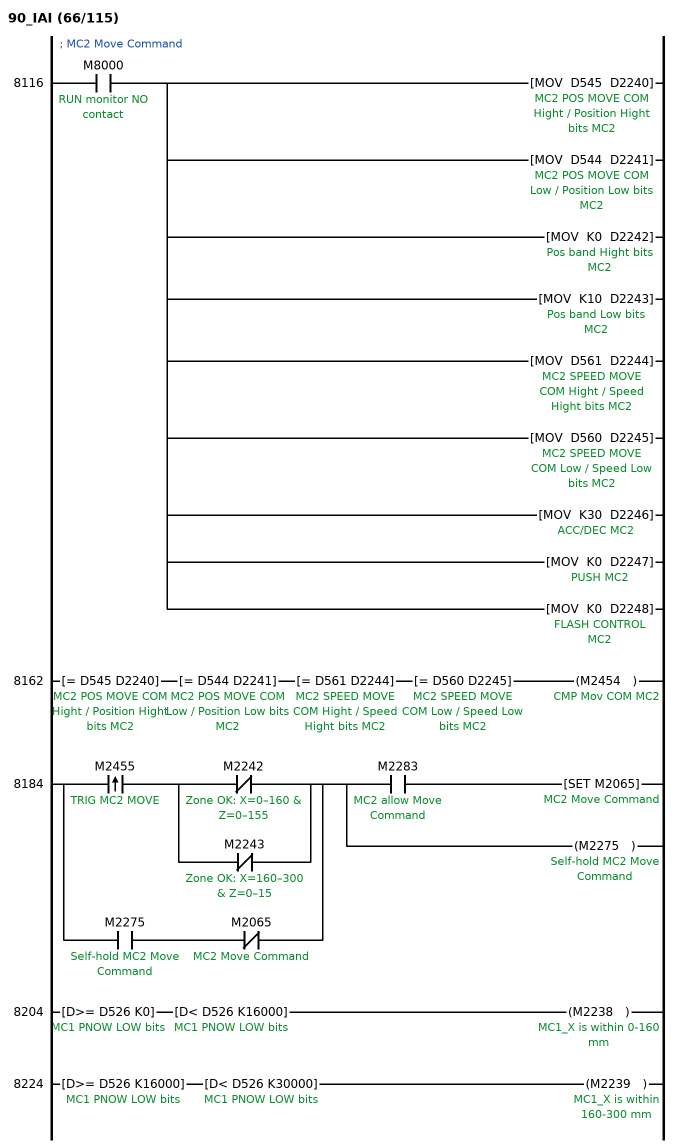
[picture p168: ladder of 90_IAI, rungs at steps 8116 to 8224]
; MC2 Move Command
8116  LD      M8000  ; RUN monitor NO contact
      MOV     D545 D2240  ; MC2 POS MOVE COM Hight / Position Hight bits MC2
      MOV     D544 D2241  ; MC2 POS MOVE COM Low / Position Low bits MC2
      MOV     K0 D2242  ; Pos band Hight bits MC2
      MOV     K10 D2243  ; Pos band Low bits MC2
      MOV     D561 D2244  ; MC2 SPEED MOVE COM Hight / Speed Hight bits MC2
      MOV     D560 D2245  ; MC2 SPEED MOVE COM Low / Speed Low bits MC2
      MOV     K30 D2246  ; ACC/DEC MC2
      MOV     K0 D2247  ; PUSH MC2
      MOV     K0 D2248  ; FLASH CONTROL MC2
8162  LD=     D545 D2240  ; MC2 POS MOVE COM Hight / Position Hight bits MC2
      AND=    D544 D2241  ; MC2 POS MOVE COM Low / Position Low bits MC2
      AND=    D561 D2244  ; MC2 SPEED MOVE COM Hight / Speed Hight bits MC2
      AND=    D560 D2245  ; MC2 SPEED MOVE COM Low / Speed Low bits MC2
      OUT     M2454  ; CMP Mov COM MC2
8184  LDP     M2455  ; TRIG MC2 MOVE
      LDI     M2242  ; Zone OK: X=0–160 & Z=0–155
      ORI     M2243  ; Zone OK: X=160–300 & Z=0–15
      ANB
      LD      M2275  ; Self-hold MC2 Move Command
      ANI     M2065  ; MC2 Move Command
      ORB
      MPS
      AND     M2283  ; MC2 allow Move Command
      SET     M2065  ; MC2 Move Command
      MPP
      OUT     M2275  ; Self-hold MC2 Move Command
8204  LDD>=   D526 K0  ; MC1 PNOW LOW bits
      ANDD<   D526 K16000  ; MC1 PNOW LOW bits
      OUT     M2238  ; MC1_X is within 0-160 mm
8224  LDD>=   D526 K16000  ; MC1 PNOW LOW bits
      ANDD<   D526 K30000  ; MC1 PNOW LOW bits
      OUT     M2239  ; MC1_X is within 160-300 mm
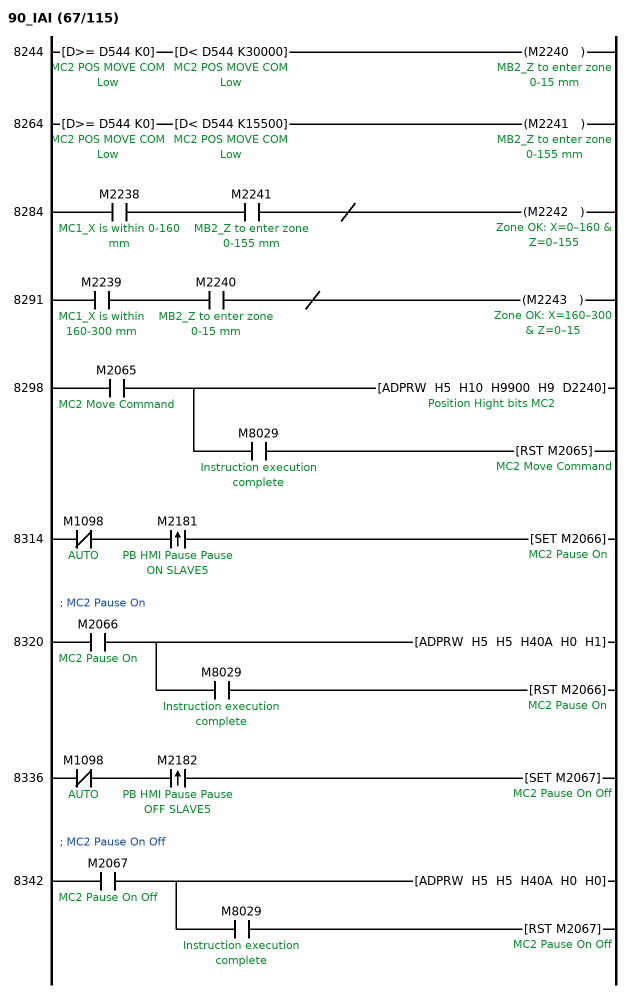
8244  LDD>=   D544 K0  ; MC2 POS MOVE COM Low
      ANDD<   D544 K30000  ; MC2 POS MOVE COM Low
      OUT     M2240  ; MB2_Z to enter zone 0-15 mm
8264  LDD>=   D544 K0  ; MC2 POS MOVE COM Low
      ANDD<   D544 K15500  ; MC2 POS MOVE COM Low
      OUT     M2241  ; MB2_Z to enter zone 0-155 mm
8284  LD      M2238  ; MC1_X is within 0-160 mm
      AND     M2241  ; MB2_Z to enter zone 0-155 mm
      INV
      OUT     M2242  ; Zone OK: X=0–160 & Z=0–155
8291  LD      M2239  ; MC1_X is within 160-300 mm
      AND     M2240  ; MB2_Z to enter zone 0-15 mm
      INV
      OUT     M2243  ; Zone OK: X=160–300 & Z=0–15
8298  LD      M2065  ; MC2 Move Command
      ADPRW   H5 H10 H9900 H9 D2240
      AND     M8029  ; Instruction execution complete
      RST     M2065  ; MC2 Move Command
8314  LDI     M1098  ; AUTO
      ANDP    M2181  ; PB HMI Pause Pause ON SLAVE5
      SET     M2066  ; MC2 Pause On
; MC2 Pause On
8320  LD      M2066  ; MC2 Pause On
      ADPRW   H5 H5 H40A H0 H1
      AND     M8029  ; Instruction execution complete
      RST     M2066  ; MC2 Pause On
8336  LDI     M1098  ; AUTO
      ANDP    M2182  ; PB HMI Pause Pause OFF SLAVE5
      SET     M2067  ; MC2 Pause On Off
; MC2 Pause On Off
8342  LD      M2067  ; MC2 Pause On Off
      ADPRW   H5 H5 H40A H0 H0
      AND     M8029  ; Instruction execution complete
      RST     M2067  ; MC2 Pause On Off
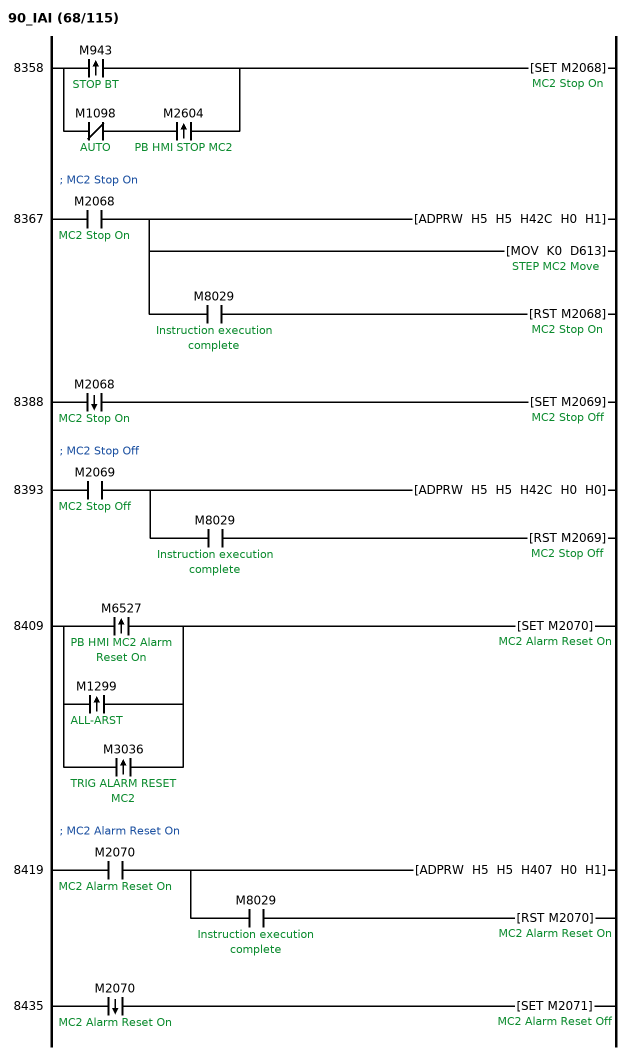
8358  LDP     M943  ; STOP BT
      LDI     M1098  ; AUTO
      ANDP    M2604  ; PB HMI STOP MC2
      ORB
      SET     M2068  ; MC2 Stop On
; MC2 Stop On
8367  LD      M2068  ; MC2 Stop On
      ADPRW   H5 H5 H42C H0 H1
      MOV     K0 D613  ; STEP MC2 Move
      AND     M8029  ; Instruction execution complete
      RST     M2068  ; MC2 Stop On
8388  LDF     M2068  ; MC2 Stop On
      SET     M2069  ; MC2 Stop Off
; MC2 Stop Off
8393  LD      M2069  ; MC2 Stop Off
      ADPRW   H5 H5 H42C H0 H0
      AND     M8029  ; Instruction execution complete
      RST     M2069  ; MC2 Stop Off
8409  LDP     M6527  ; PB HMI MC2 Alarm Reset On
      ORP     M1299  ; ALL-ARST
      ORP     M3036  ; TRIG ALARM RESET MC2
      SET     M2070  ; MC2 Alarm Reset On
; MC2 Alarm Reset On
8419  LD      M2070  ; MC2 Alarm Reset On
      ADPRW   H5 H5 H407 H0 H1
      AND     M8029  ; Instruction execution complete
      RST     M2070  ; MC2 Alarm Reset On
8435  LDF     M2070  ; MC2 Alarm Reset On
      SET     M2071  ; MC2 Alarm Reset Off
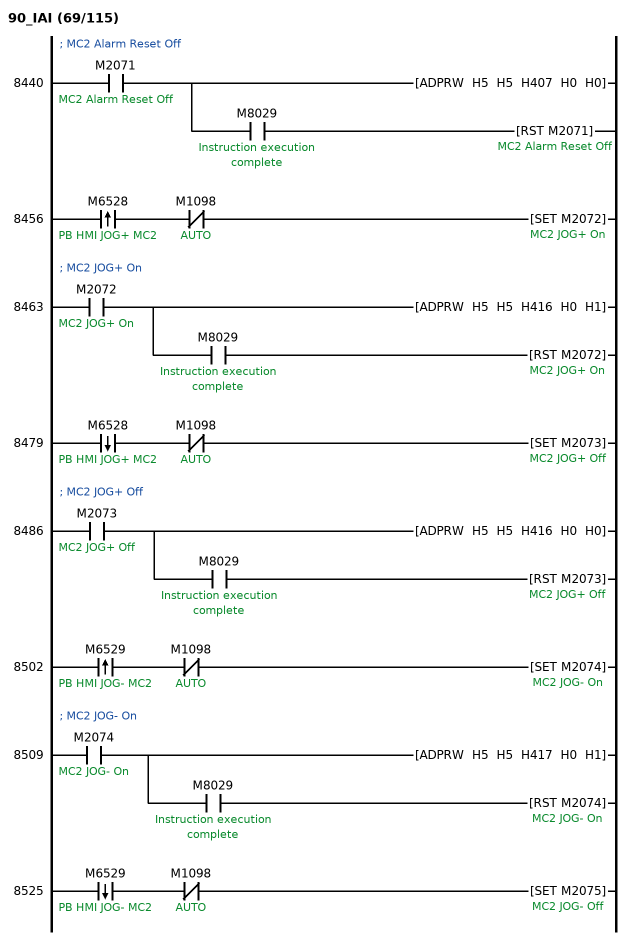
; MC2 Alarm Reset Off
8440  LD      M2071  ; MC2 Alarm Reset Off
      ADPRW   H5 H5 H407 H0 H0
      AND     M8029  ; Instruction execution complete
      RST     M2071  ; MC2 Alarm Reset Off
8456  LDP     M6528  ; PB HMI JOG+ MC2
      ANI     M1098  ; AUTO
      SET     M2072  ; MC2 JOG+ On
; MC2 JOG+ On
8463  LD      M2072  ; MC2 JOG+ On
      ADPRW   H5 H5 H416 H0 H1
      AND     M8029  ; Instruction execution complete
      RST     M2072  ; MC2 JOG+ On
8479  LDF     M6528  ; PB HMI JOG+ MC2
      ANI     M1098  ; AUTO
      SET     M2073  ; MC2 JOG+ Off
; MC2 JOG+ Off
8486  LD      M2073  ; MC2 JOG+ Off
      ADPRW   H5 H5 H416 H0 H0
      AND     M8029  ; Instruction execution complete
      RST     M2073  ; MC2 JOG+ Off
8502  LDP     M6529  ; PB HMI JOG- MC2
      ANI     M1098  ; AUTO
      SET     M2074  ; MC2 JOG- On
; MC2 JOG- On
8509  LD      M2074  ; MC2 JOG- On
      ADPRW   H5 H5 H417 H0 H1
      AND     M8029  ; Instruction execution complete
      RST     M2074  ; MC2 JOG- On
8525  LDF     M6529  ; PB HMI JOG- MC2
      ANI     M1098  ; AUTO
      SET     M2075  ; MC2 JOG- Off
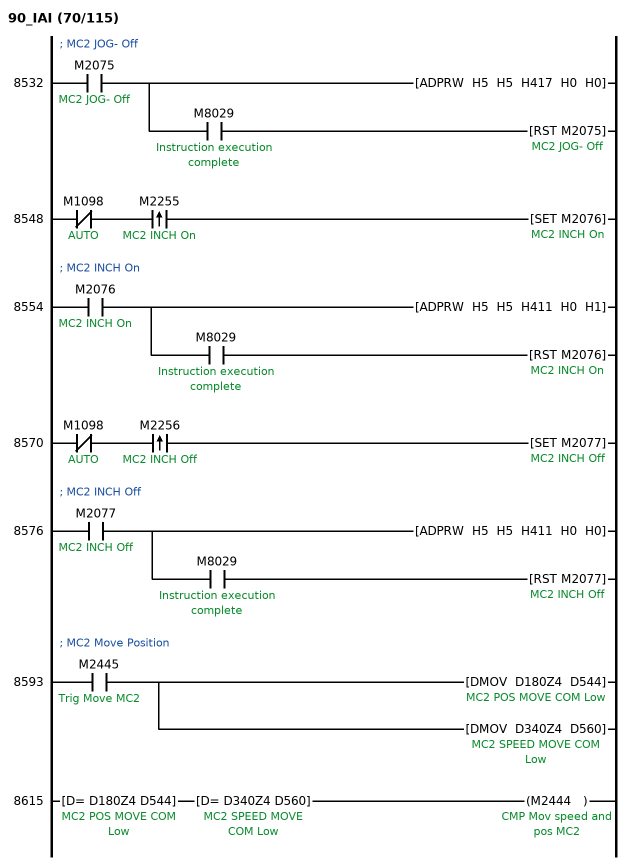
; MC2 JOG- Off
8532  LD      M2075  ; MC2 JOG- Off
      ADPRW   H5 H5 H417 H0 H0
      AND     M8029  ; Instruction execution complete
      RST     M2075  ; MC2 JOG- Off
8548  LDI     M1098  ; AUTO
      ANDP    M2255  ; MC2 INCH On
      SET     M2076  ; MC2 INCH On
; MC2 INCH On
8554  LD      M2076  ; MC2 INCH On
      ADPRW   H5 H5 H411 H0 H1
      AND     M8029  ; Instruction execution complete
      RST     M2076  ; MC2 INCH On
8570  LDI     M1098  ; AUTO
      ANDP    M2256  ; MC2 INCH Off
      SET     M2077  ; MC2 INCH Off
; MC2 INCH Off
8576  LD      M2077  ; MC2 INCH Off
      ADPRW   H5 H5 H411 H0 H0
      AND     M8029  ; Instruction execution complete
      RST     M2077  ; MC2 INCH Off
; MC2 Move Position
8593  LD      M2445  ; Trig Move MC2
      DMOV    D180Z4 D544
        [note] Position
      DMOV    D340Z4 D560
        [note] Speed
8615  LDD=    D180Z4 D544  ; MC2 POS MOVE COM Low
      ANDD=   D340Z4 D560  ; MC2 SPEED MOVE COM Low
      OUT     M2444  ; CMP Mov speed and pos MC2
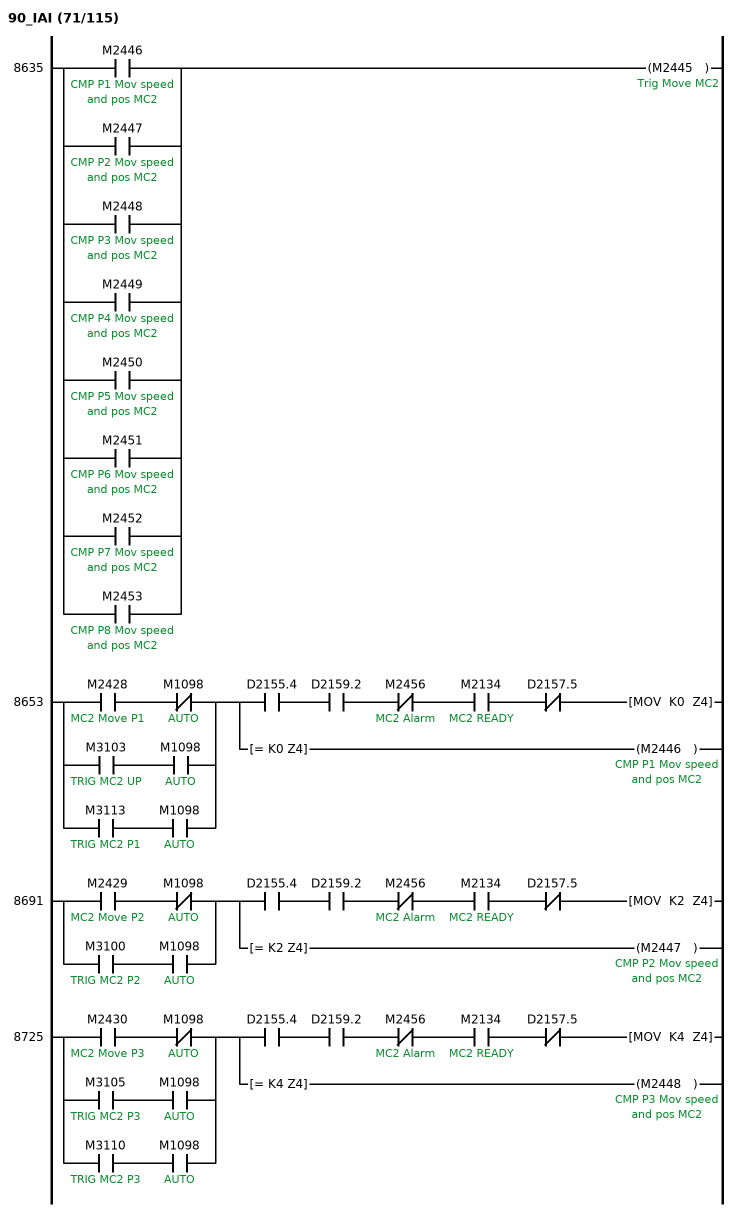
8635  LD      M2446  ; CMP P1 Mov speed and pos MC2
      OR      M2447  ; CMP P2 Mov speed and pos MC2
      OR      M2448  ; CMP P3 Mov speed and pos MC2
      OR      M2449  ; CMP P4 Mov speed and pos MC2
      OR      M2450  ; CMP P5 Mov speed and pos MC2
      OR      M2451  ; CMP P6 Mov speed and pos MC2
      OR      M2452  ; CMP P7 Mov speed and pos MC2
      OR      M2453  ; CMP P8 Mov speed and pos MC2
      OUT     M2445  ; Trig Move MC2
8653  LD      M2428  ; MC2 Move P1
      ANI     M1098  ; AUTO
      LD      M3103  ; TRIG MC2 UP
      AND     M1098  ; AUTO
      ORB
      LD      M3113  ; TRIG MC2 P1
      AND     M1098  ; AUTO
      ORB
      MPS
      AND     D2155.4
      AND     D2159.2
      ANI     M2456  ; MC2 Alarm
      AND     M2134  ; MC2 READY
      ANI     D2157.5
      MOV     K0 Z4
      MPP
      AND=    K0 Z4
      OUT     M2446  ; CMP P1 Mov speed and pos MC2
8691  LD      M2429  ; MC2 Move P2
      ANI     M1098  ; AUTO
      LD      M3100  ; TRIG MC2 P2
      AND     M1098  ; AUTO
      ORB
      MPS
      AND     D2155.4
      AND     D2159.2
      ANI     M2456  ; MC2 Alarm
      AND     M2134  ; MC2 READY
      ANI     D2157.5
      MOV     K2 Z4
      MPP
      AND=    K2 Z4
      OUT     M2447  ; CMP P2 Mov speed and pos MC2
8725  LD      M2430  ; MC2 Move P3
      ANI     M1098  ; AUTO
      LD      M3105  ; TRIG MC2 P3
      AND     M1098  ; AUTO
      ORB
      LD      M3110  ; TRIG MC2 P3
      AND     M1098  ; AUTO
      ORB
      MPS
      AND     D2155.4
      AND     D2159.2
      ANI     M2456  ; MC2 Alarm
      AND     M2134  ; MC2 READY
      ANI     D2157.5
      MOV     K4 Z4
      MPP
      AND=    K4 Z4
      OUT     M2448  ; CMP P3 Mov speed and pos MC2
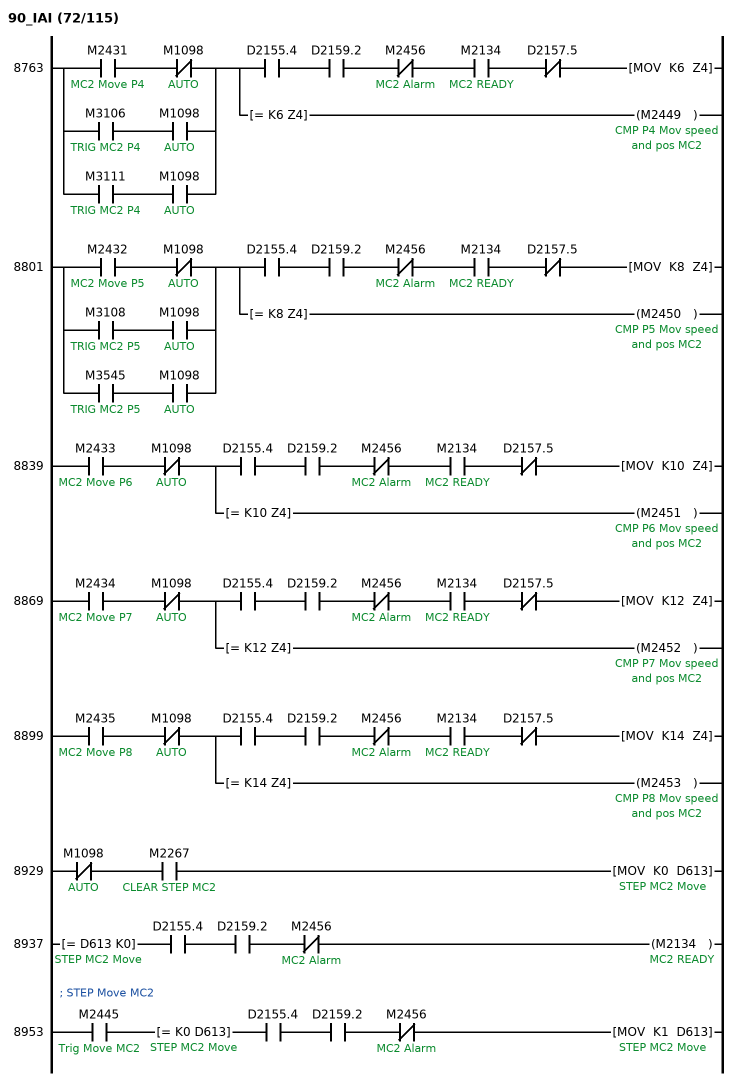
8763  LD      M2431  ; MC2 Move P4
      ANI     M1098  ; AUTO
      LD      M3106  ; TRIG MC2 P4
      AND     M1098  ; AUTO
      ORB
      LD      M3111  ; TRIG MC2 P4
      AND     M1098  ; AUTO
      ORB
      MPS
      AND     D2155.4
      AND     D2159.2
      ANI     M2456  ; MC2 Alarm
      AND     M2134  ; MC2 READY
      ANI     D2157.5
      MOV     K6 Z4
      MPP
      AND=    K6 Z4
      OUT     M2449  ; CMP P4 Mov speed and pos MC2
8801  LD      M2432  ; MC2 Move P5
      ANI     M1098  ; AUTO
      LD      M3108  ; TRIG MC2 P5
      AND     M1098  ; AUTO
      ORB
      LD      M3545  ; TRIG MC2 P5
      AND     M1098  ; AUTO
      ORB
      MPS
      AND     D2155.4
      AND     D2159.2
      ANI     M2456  ; MC2 Alarm
      AND     M2134  ; MC2 READY
      ANI     D2157.5
      MOV     K8 Z4
      MPP
      AND=    K8 Z4
      OUT     M2450  ; CMP P5 Mov speed and pos MC2
8839  LD      M2433  ; MC2 Move P6
      ANI     M1098  ; AUTO
      MPS
      AND     D2155.4
      AND     D2159.2
      ANI     M2456  ; MC2 Alarm
      AND     M2134  ; MC2 READY
      ANI     D2157.5
      MOV     K10 Z4
      MPP
      AND=    K10 Z4
      OUT     M2451  ; CMP P6 Mov speed and pos MC2
8869  LD      M2434  ; MC2 Move P7
      ANI     M1098  ; AUTO
      MPS
      AND     D2155.4
      AND     D2159.2
      ANI     M2456  ; MC2 Alarm
      AND     M2134  ; MC2 READY
      ANI     D2157.5
      MOV     K12 Z4
      MPP
      AND=    K12 Z4
      OUT     M2452  ; CMP P7 Mov speed and pos MC2
8899  LD      M2435  ; MC2 Move P8
      ANI     M1098  ; AUTO
      MPS
      AND     D2155.4
      AND     D2159.2
      ANI     M2456  ; MC2 Alarm
      AND     M2134  ; MC2 READY
      ANI     D2157.5
      MOV     K14 Z4
      MPP
      AND=    K14 Z4
      OUT     M2453  ; CMP P8 Mov speed and pos MC2
8929  LDI     M1098  ; AUTO
      AND     M2267  ; CLEAR STEP MC2
      MOV     K0 D613
8937  LD=     D613 K0  ; STEP MC2 Move
      AND     D2155.4
      AND     D2159.2
      ANI     M2456  ; MC2 Alarm
      OUT     M2134  ; MC2 READY
; STEP Move MC2
8953  LD      M2445  ; Trig Move MC2
      AND=    K0 D613  ; STEP MC2 Move
      AND     D2155.4
      AND     D2159.2
      ANI     M2456  ; MC2 Alarm
      MOV     K1 D613
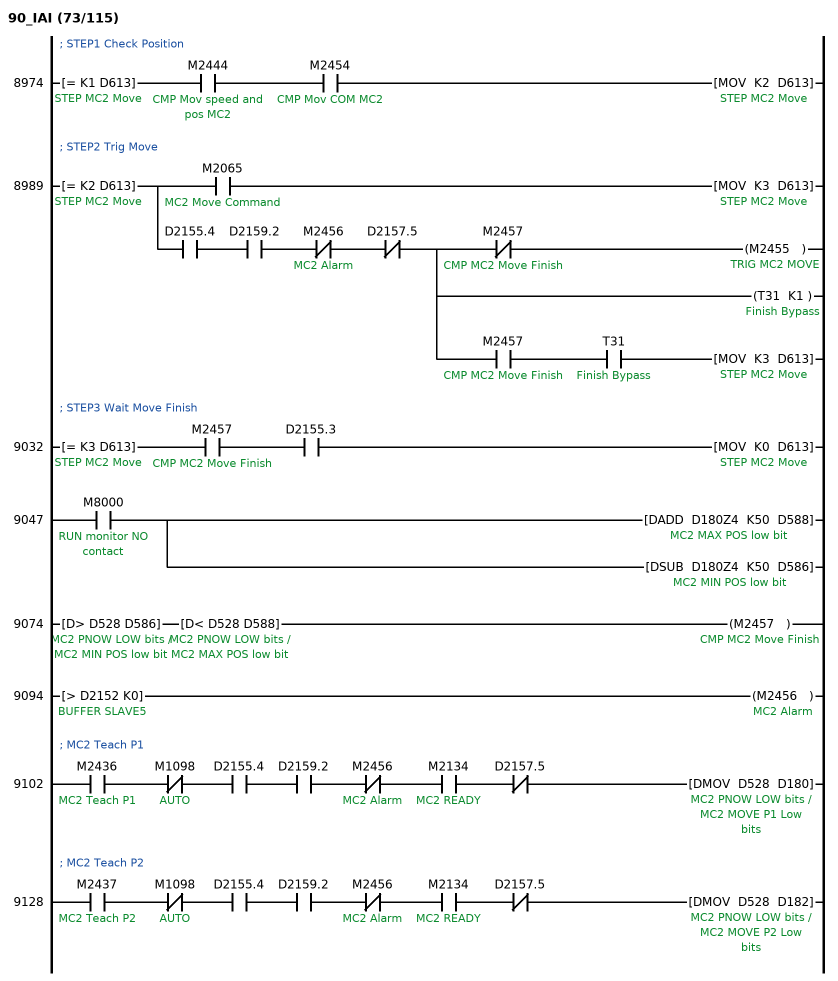
; STEP1 Check Position
8974  LD=     K1 D613  ; STEP MC2 Move
      AND     M2444  ; CMP Mov speed and pos MC2
      AND     M2454  ; CMP Mov COM MC2
      MOV     K2 D613
; STEP2 Trig Move
8989  LD=     K2 D613  ; STEP MC2 Move
      MPS
      AND     M2065  ; MC2 Move Command
      MOV     K3 D613
      MPP
      AND     D2155.4
      AND     D2159.2
      ANI     M2456  ; MC2 Alarm
      ANI     D2157.5
      MPS
      ANI     M2457  ; CMP MC2 Move Finish
      OUT     M2455  ; TRIG MC2 MOVE
      MPP
      OUT     T31 K1  ; Finish Bypass
      AND     M2457  ; CMP MC2 Move Finish
      AND     T31  ; Finish Bypass
      MOV     K3 D613
; STEP3 Wait Move Finish
9032  LD=     K3 D613  ; STEP MC2 Move
      AND     M2457  ; CMP MC2 Move Finish
      AND     D2155.3
      MOV     K0 D613
9047  LD      M8000  ; RUN monitor NO contact
      DADD    D180Z4 K50 D588  ; MC2 MAX POS low bit
      DSUB    D180Z4 K50 D586  ; MC2 MIN POS low bit
9074  LDD>    D528 D586  ; MC2 PNOW LOW bits / MC2 MIN POS low bit
      ANDD<   D528 D588  ; MC2 PNOW LOW bits / MC2 MAX POS low bit
      OUT     M2457  ; CMP MC2 Move Finish
9094  LD>     D2152 K0  ; BUFFER SLAVE5
      OUT     M2456  ; MC2 Alarm
; MC2 Teach P1
9102  LD      M2436  ; MC2 Teach P1
      ANI     M1098  ; AUTO
      AND     D2155.4
      AND     D2159.2
      ANI     M2456  ; MC2 Alarm
      AND     M2134  ; MC2 READY
      ANI     D2157.5
      DMOV    D528 D180  ; MC2 MOVE P1 Low bits
; MC2 Teach P2
9128  LD      M2437  ; MC2 Teach P2
      ANI     M1098  ; AUTO
      AND     D2155.4
      AND     D2159.2
      ANI     M2456  ; MC2 Alarm
      AND     M2134  ; MC2 READY
      ANI     D2157.5
      DMOV    D528 D182  ; MC2 MOVE P2 Low bits
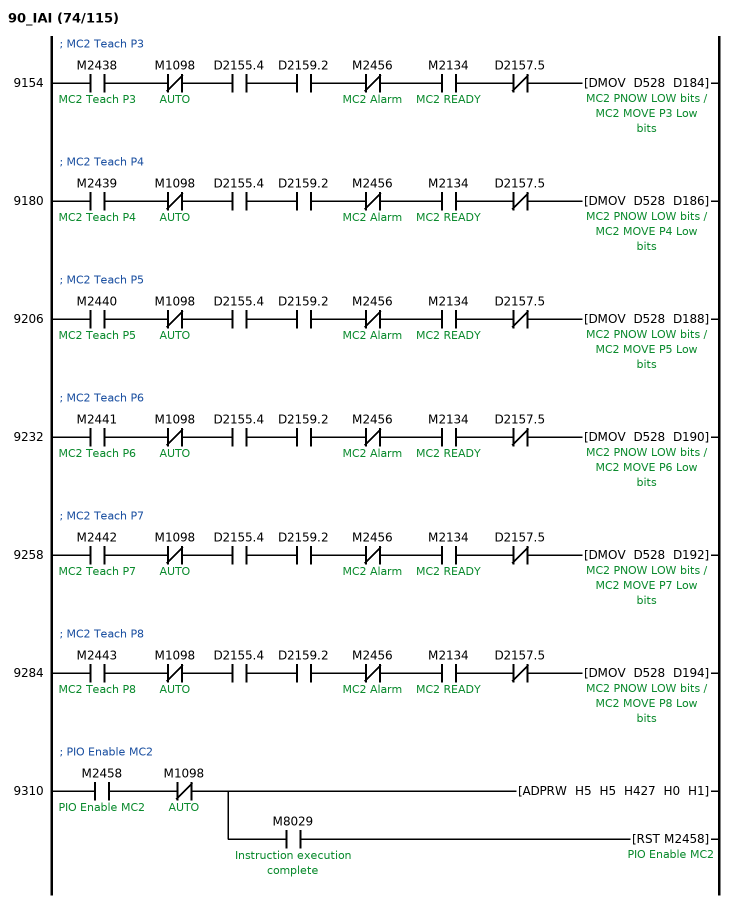
; MC2 Teach P3
9154  LD      M2438  ; MC2 Teach P3
      ANI     M1098  ; AUTO
      AND     D2155.4
      AND     D2159.2
      ANI     M2456  ; MC2 Alarm
      AND     M2134  ; MC2 READY
      ANI     D2157.5
      DMOV    D528 D184  ; MC2 MOVE P3 Low bits
; MC2 Teach P4
9180  LD      M2439  ; MC2 Teach P4
      ANI     M1098  ; AUTO
      AND     D2155.4
      AND     D2159.2
      ANI     M2456  ; MC2 Alarm
      AND     M2134  ; MC2 READY
      ANI     D2157.5
      DMOV    D528 D186  ; MC2 MOVE P4 Low bits
; MC2 Teach P5
9206  LD      M2440  ; MC2 Teach P5
      ANI     M1098  ; AUTO
      AND     D2155.4
      AND     D2159.2
      ANI     M2456  ; MC2 Alarm
      AND     M2134  ; MC2 READY
      ANI     D2157.5
      DMOV    D528 D188  ; MC2 MOVE P5 Low bits
; MC2 Teach P6
9232  LD      M2441  ; MC2 Teach P6
      ANI     M1098  ; AUTO
      AND     D2155.4
      AND     D2159.2
      ANI     M2456  ; MC2 Alarm
      AND     M2134  ; MC2 READY
      ANI     D2157.5
      DMOV    D528 D190  ; MC2 MOVE P6 Low bits
; MC2 Teach P7
9258  LD      M2442  ; MC2 Teach P7
      ANI     M1098  ; AUTO
      AND     D2155.4
      AND     D2159.2
      ANI     M2456  ; MC2 Alarm
      AND     M2134  ; MC2 READY
      ANI     D2157.5
      DMOV    D528 D192  ; MC2 MOVE P7 Low bits
; MC2 Teach P8
9284  LD      M2443  ; MC2 Teach P8
      ANI     M1098  ; AUTO
      AND     D2155.4
      AND     D2159.2
      ANI     M2456  ; MC2 Alarm
      AND     M2134  ; MC2 READY
      ANI     D2157.5
      DMOV    D528 D194  ; MC2 MOVE P8 Low bits
; PIO Enable MC2
9310  LD      M2458  ; PIO Enable MC2
      ANI     M1098  ; AUTO
      ADPRW   H5 H5 H427 H0 H1
      AND     M8029  ; Instruction execution complete
      RST     M2458  ; PIO Enable MC2
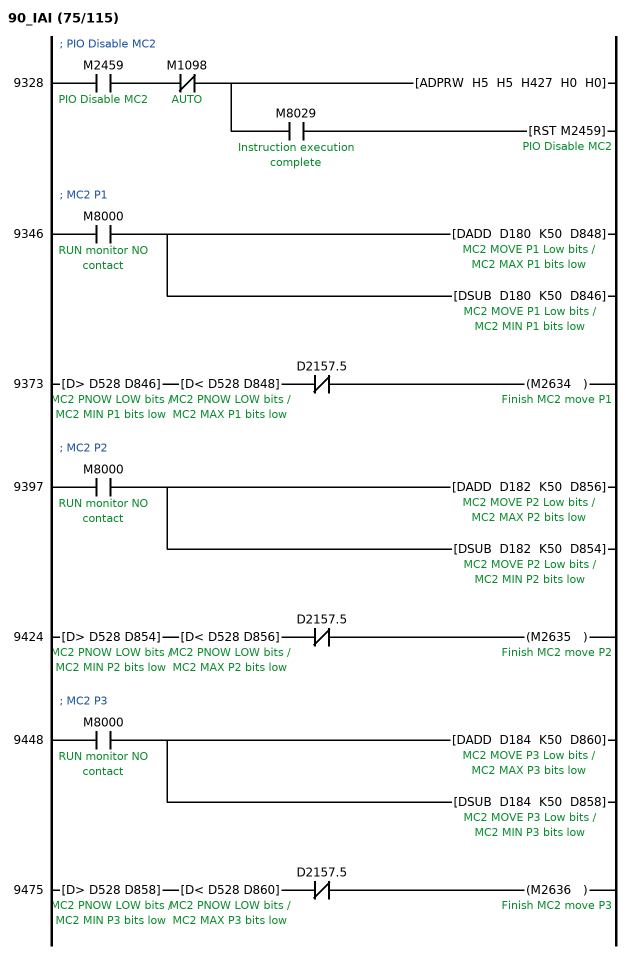
; PIO Disable MC2
9328  LD      M2459  ; PIO Disable MC2
      ANI     M1098  ; AUTO
      ADPRW   H5 H5 H427 H0 H0
      AND     M8029  ; Instruction execution complete
      RST     M2459  ; PIO Disable MC2
; MC2 P1
9346  LD      M8000  ; RUN monitor NO contact
      DADD    D180 K50 D848  ; MC2 MAX P1 bits low
      DSUB    D180 K50 D846  ; MC2 MIN P1 bits low
9373  LDD>    D528 D846  ; MC2 PNOW LOW bits / MC2 MIN P1 bits low
      ANDD<   D528 D848  ; MC2 PNOW LOW bits / MC2 MAX P1 bits low
      ANI     D2157.5
      OUT     M2634  ; Finish MC2 move P1
; MC2 P2
9397  LD      M8000  ; RUN monitor NO contact
      DADD    D182 K50 D856  ; MC2 MAX P2 bits low
      DSUB    D182 K50 D854  ; MC2 MIN P2 bits low
9424  LDD>    D528 D854  ; MC2 PNOW LOW bits / MC2 MIN P2 bits low
      ANDD<   D528 D856  ; MC2 PNOW LOW bits / MC2 MAX P2 bits low
      ANI     D2157.5
      OUT     M2635  ; Finish MC2 move P2
; MC2 P3
9448  LD      M8000  ; RUN monitor NO contact
      DADD    D184 K50 D860  ; MC2 MAX P3 bits low
      DSUB    D184 K50 D858  ; MC2 MIN P3 bits low
9475  LDD>    D528 D858  ; MC2 PNOW LOW bits / MC2 MIN P3 bits low
      ANDD<   D528 D860  ; MC2 PNOW LOW bits / MC2 MAX P3 bits low
      ANI     D2157.5
      OUT     M2636  ; Finish MC2 move P3
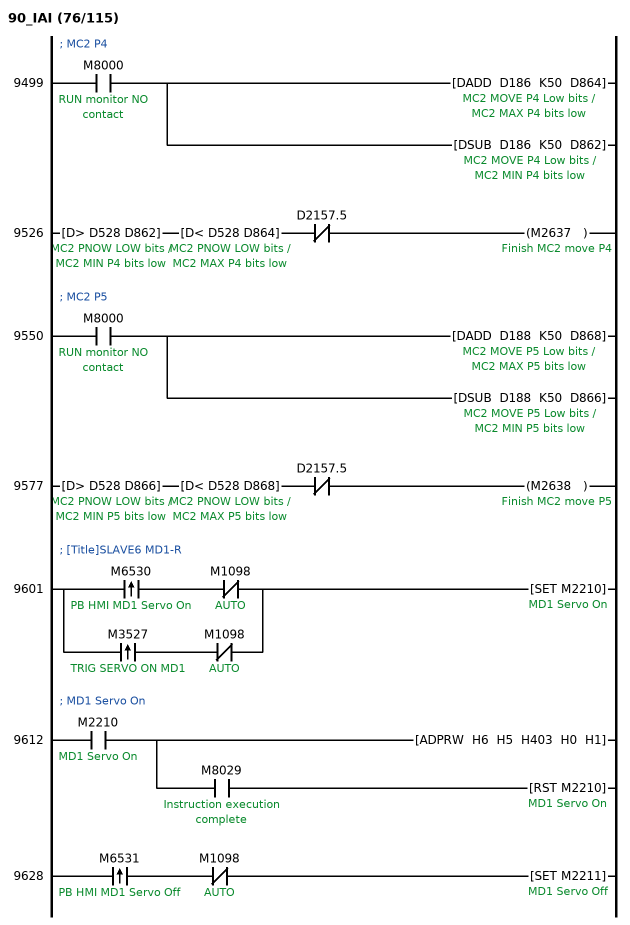
; MC2 P4
9499  LD      M8000  ; RUN monitor NO contact
      DADD    D186 K50 D864  ; MC2 MAX P4 bits low
      DSUB    D186 K50 D862  ; MC2 MIN P4 bits low
9526  LDD>    D528 D862  ; MC2 PNOW LOW bits / MC2 MIN P4 bits low
      ANDD<   D528 D864  ; MC2 PNOW LOW bits / MC2 MAX P4 bits low
      ANI     D2157.5
      OUT     M2637  ; Finish MC2 move P4
; MC2 P5
9550  LD      M8000  ; RUN monitor NO contact
      DADD    D188 K50 D868  ; MC2 MAX P5 bits low
      DSUB    D188 K50 D866  ; MC2 MIN P5 bits low
9577  LDD>    D528 D866  ; MC2 PNOW LOW bits / MC2 MIN P5 bits low
      ANDD<   D528 D868  ; MC2 PNOW LOW bits / MC2 MAX P5 bits low
      ANI     D2157.5
      OUT     M2638  ; Finish MC2 move P5
; [Title]SLAVE6 MD1-R
9601  LDP     M6530  ; PB HMI MD1 Servo On
      ANI     M1098  ; AUTO
      LDP     M3527  ; TRIG SERVO ON MD1
      ANI     M1098  ; AUTO
      ORB
      SET     M2210  ; MD1 Servo On
; MD1 Servo On
9612  LD      M2210  ; MD1 Servo On
      ADPRW   H6 H5 H403 H0 H1
      AND     M8029  ; Instruction execution complete
      RST     M2210  ; MD1 Servo On
9628  LDP     M6531  ; PB HMI MD1 Servo Off
      ANI     M1098  ; AUTO
      SET     M2211  ; MD1 Servo Off
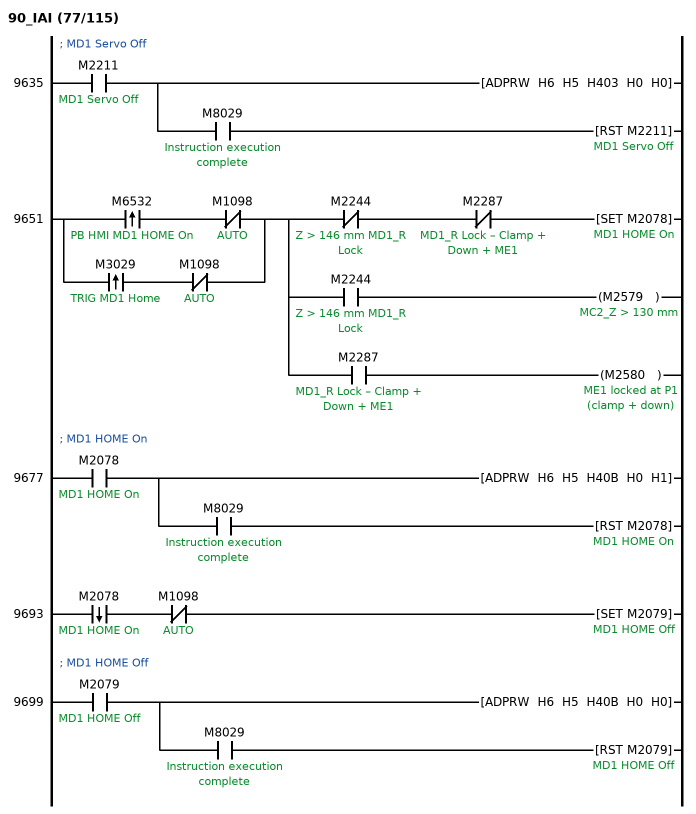
; MD1 Servo Off
9635  LD      M2211  ; MD1 Servo Off
      ADPRW   H6 H5 H403 H0 H0
      AND     M8029  ; Instruction execution complete
      RST     M2211  ; MD1 Servo Off
9651  LDP     M6532  ; PB HMI MD1 HOME On
      ANI     M1098  ; AUTO
      LDP     M3029  ; TRIG MD1 Home
      ANI     M1098  ; AUTO
      ORB
      MPS
      ANI     M2244  ; Z > 146 mm MD1_R Lock
      ANI     M2287  ; MD1_R Lock – Clamp + Down + ME1
      SET     M2078  ; MD1 HOME On
      MRD
      AND     M2244  ; Z > 146 mm MD1_R Lock
      OUT     M2579  ; MC2_Z > 130 mm
      MPP
      AND     M2287  ; MD1_R Lock – Clamp + Down + ME1
      OUT     M2580  ; ME1 locked at P1 (clamp + down)
; MD1 HOME On
9677  LD      M2078  ; MD1 HOME On
      ADPRW   H6 H5 H40B H0 H1
      AND     M8029  ; Instruction execution complete
      RST     M2078  ; MD1 HOME On
9693  LDF     M2078  ; MD1 HOME On
      ANI     M1098  ; AUTO
      SET     M2079  ; MD1 HOME Off
; MD1 HOME Off
9699  LD      M2079  ; MD1 HOME Off
      ADPRW   H6 H5 H40B H0 H0
      AND     M8029  ; Instruction execution complete
      RST     M2079  ; MD1 HOME Off
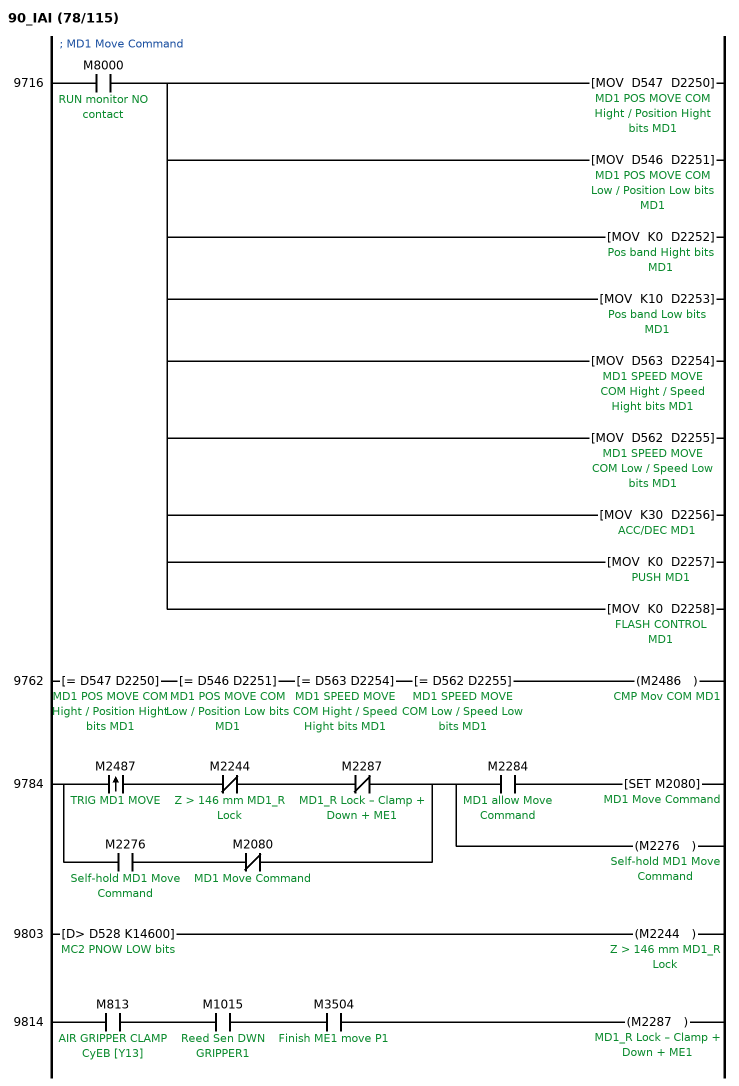
; MD1 Move Command
9716  LD      M8000  ; RUN monitor NO contact
      MOV     D547 D2250  ; MD1 POS MOVE COM Hight / Position Hight bits MD1
      MOV     D546 D2251  ; MD1 POS MOVE COM Low / Position Low bits MD1
      MOV     K0 D2252  ; Pos band Hight bits MD1
      MOV     K10 D2253  ; Pos band Low bits MD1
      MOV     D563 D2254  ; MD1 SPEED MOVE COM Hight / Speed Hight bits MD1
      MOV     D562 D2255  ; MD1 SPEED MOVE COM Low / Speed Low bits MD1
      MOV     K30 D2256  ; ACC/DEC MD1
      MOV     K0 D2257  ; PUSH MD1
      MOV     K0 D2258  ; FLASH CONTROL MD1
9762  LD=     D547 D2250  ; MD1 POS MOVE COM Hight / Position Hight bits MD1
      AND=    D546 D2251  ; MD1 POS MOVE COM Low / Position Low bits MD1
      AND=    D563 D2254  ; MD1 SPEED MOVE COM Hight / Speed Hight bits MD1
      AND=    D562 D2255  ; MD1 SPEED MOVE COM Low / Speed Low bits MD1
      OUT     M2486  ; CMP Mov COM MD1
9784  LDP     M2487  ; TRIG MD1 MOVE
      ANI     M2244  ; Z > 146 mm MD1_R Lock
      ANI     M2287  ; MD1_R Lock – Clamp + Down + ME1
      LD      M2276  ; Self-hold MD1 Move Command
      ANI     M2080  ; MD1 Move Command
      ORB
      MPS
      AND     M2284  ; MD1 allow Move Command
      SET     M2080  ; MD1 Move Command
      MPP
      OUT     M2276  ; Self-hold MD1 Move Command
9803  LDD>    D528 K14600  ; MC2 PNOW LOW bits
      OUT     M2244  ; Z > 146 mm MD1_R Lock
9814  LD      M813  ; AIR GRIPPER CLAMP CyEB [Y13]
      AND     M1015  ; Reed Sen DWN GRIPPER1
      AND     M3504  ; Finish ME1 move P1
      OUT     M2287  ; MD1_R Lock – Clamp + Down + ME1
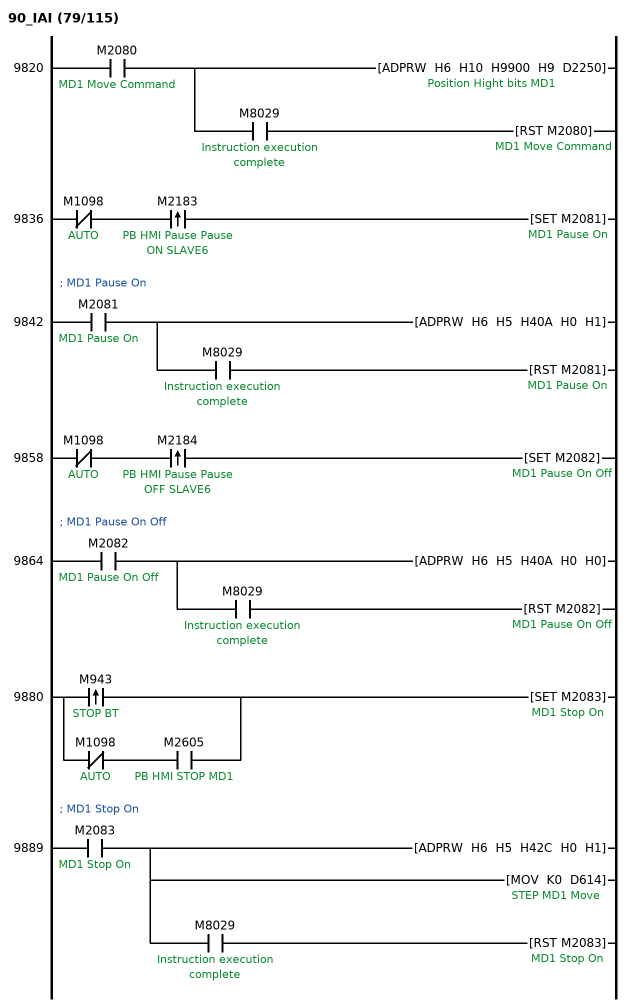
9820  LD      M2080  ; MD1 Move Command
      ADPRW   H6 H10 H9900 H9 D2250
      AND     M8029  ; Instruction execution complete
      RST     M2080  ; MD1 Move Command
9836  LDI     M1098  ; AUTO
      ANDP    M2183  ; PB HMI Pause Pause ON SLAVE6
      SET     M2081  ; MD1 Pause On
; MD1 Pause On
9842  LD      M2081  ; MD1 Pause On
      ADPRW   H6 H5 H40A H0 H1
      AND     M8029  ; Instruction execution complete
      RST     M2081  ; MD1 Pause On
9858  LDI     M1098  ; AUTO
      ANDP    M2184  ; PB HMI Pause Pause OFF SLAVE6
      SET     M2082  ; MD1 Pause On Off
; MD1 Pause On Off
9864  LD      M2082  ; MD1 Pause On Off
      ADPRW   H6 H5 H40A H0 H0
      AND     M8029  ; Instruction execution complete
      RST     M2082  ; MD1 Pause On Off
9880  LDP     M943  ; STOP BT
      LDI     M1098  ; AUTO
      AND     M2605  ; PB HMI STOP MD1
      ORB
      SET     M2083  ; MD1 Stop On
; MD1 Stop On
9889  LD      M2083  ; MD1 Stop On
      ADPRW   H6 H5 H42C H0 H1
      MOV     K0 D614  ; STEP MD1 Move
      AND     M8029  ; Instruction execution complete
      RST     M2083  ; MD1 Stop On
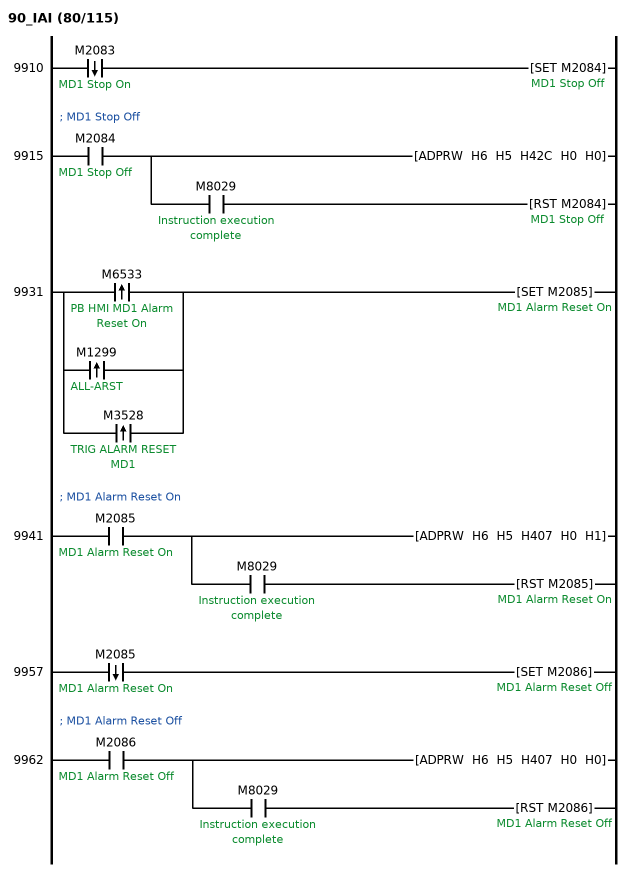
9910  LDF     M2083  ; MD1 Stop On
      SET     M2084  ; MD1 Stop Off
; MD1 Stop Off
9915  LD      M2084  ; MD1 Stop Off
      ADPRW   H6 H5 H42C H0 H0
      AND     M8029  ; Instruction execution complete
      RST     M2084  ; MD1 Stop Off
9931  LDP     M6533  ; PB HMI MD1 Alarm Reset On
      ORP     M1299  ; ALL-ARST
      ORP     M3528  ; TRIG ALARM RESET MD1
      SET     M2085  ; MD1 Alarm Reset On
; MD1 Alarm Reset On
9941  LD      M2085  ; MD1 Alarm Reset On
      ADPRW   H6 H5 H407 H0 H1
      AND     M8029  ; Instruction execution complete
      RST     M2085  ; MD1 Alarm Reset On
9957  LDF     M2085  ; MD1 Alarm Reset On
      SET     M2086  ; MD1 Alarm Reset Off
; MD1 Alarm Reset Off
9962  LD      M2086  ; MD1 Alarm Reset Off
      ADPRW   H6 H5 H407 H0 H0
      AND     M8029  ; Instruction execution complete
      RST     M2086  ; MD1 Alarm Reset Off
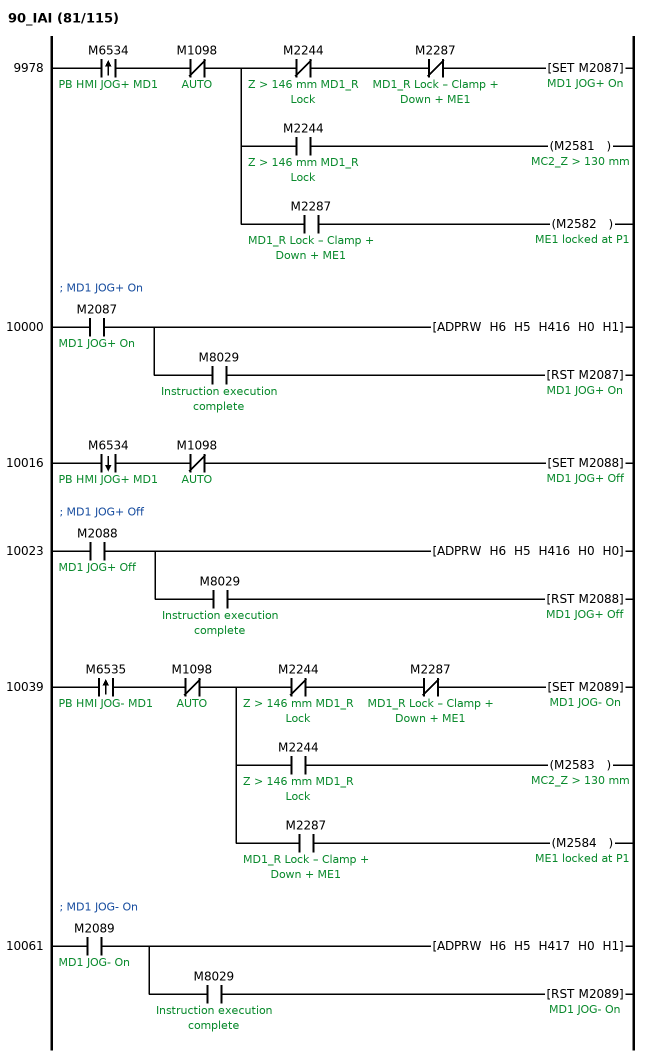
9978  LDP     M6534  ; PB HMI JOG+ MD1
      ANI     M1098  ; AUTO
      MPS
      ANI     M2244  ; Z > 146 mm MD1_R Lock
      ANI     M2287  ; MD1_R Lock – Clamp + Down + ME1
      SET     M2087  ; MD1 JOG+ On
      MRD
      AND     M2244  ; Z > 146 mm MD1_R Lock
      OUT     M2581  ; MC2_Z > 130 mm
      MPP
      AND     M2287  ; MD1_R Lock – Clamp + Down + ME1
      OUT     M2582  ; ME1 locked at P1
; MD1 JOG+ On
10000 LD      M2087  ; MD1 JOG+ On
      ADPRW   H6 H5 H416 H0 H1
      AND     M8029  ; Instruction execution complete
      RST     M2087  ; MD1 JOG+ On
10016 LDF     M6534  ; PB HMI JOG+ MD1
      ANI     M1098  ; AUTO
      SET     M2088  ; MD1 JOG+ Off
; MD1 JOG+ Off
10023 LD      M2088  ; MD1 JOG+ Off
      ADPRW   H6 H5 H416 H0 H0
      AND     M8029  ; Instruction execution complete
      RST     M2088  ; MD1 JOG+ Off
10039 LDP     M6535  ; PB HMI JOG- MD1
      ANI     M1098  ; AUTO
      MPS
      ANI     M2244  ; Z > 146 mm MD1_R Lock
      ANI     M2287  ; MD1_R Lock – Clamp + Down + ME1
      SET     M2089  ; MD1 JOG- On
      MRD
      AND     M2244  ; Z > 146 mm MD1_R Lock
      OUT     M2583  ; MC2_Z > 130 mm
      MPP
      AND     M2287  ; MD1_R Lock – Clamp + Down + ME1
      OUT     M2584  ; ME1 locked at P1
; MD1 JOG- On
10061 LD      M2089  ; MD1 JOG- On
      ADPRW   H6 H5 H417 H0 H1
      AND     M8029  ; Instruction execution complete
      RST     M2089  ; MD1 JOG- On
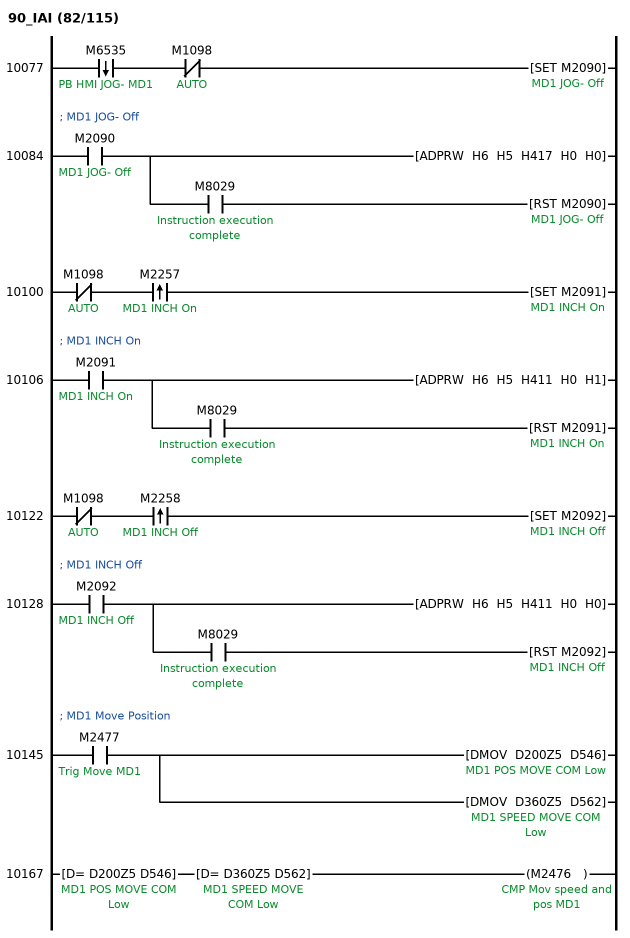
10077 LDF     M6535  ; PB HMI JOG- MD1
      ANI     M1098  ; AUTO
      SET     M2090  ; MD1 JOG- Off
; MD1 JOG- Off
10084 LD      M2090  ; MD1 JOG- Off
      ADPRW   H6 H5 H417 H0 H0
      AND     M8029  ; Instruction execution complete
      RST     M2090  ; MD1 JOG- Off
10100 LDI     M1098  ; AUTO
      ANDP    M2257  ; MD1 INCH On
      SET     M2091  ; MD1 INCH On
; MD1 INCH On
10106 LD      M2091  ; MD1 INCH On
      ADPRW   H6 H5 H411 H0 H1
      AND     M8029  ; Instruction execution complete
      RST     M2091  ; MD1 INCH On
10122 LDI     M1098  ; AUTO
      ANDP    M2258  ; MD1 INCH Off
      SET     M2092  ; MD1 INCH Off
; MD1 INCH Off
10128 LD      M2092  ; MD1 INCH Off
      ADPRW   H6 H5 H411 H0 H0
      AND     M8029  ; Instruction execution complete
      RST     M2092  ; MD1 INCH Off
; MD1 Move Position
10145 LD      M2477  ; Trig Move MD1
      DMOV    D200Z5 D546
        [note] Position
      DMOV    D360Z5 D562
        [note] Speed
10167 LDD=    D200Z5 D546  ; MD1 POS MOVE COM Low
      ANDD=   D360Z5 D562  ; MD1 SPEED MOVE COM Low
      OUT     M2476  ; CMP Mov speed and pos MD1
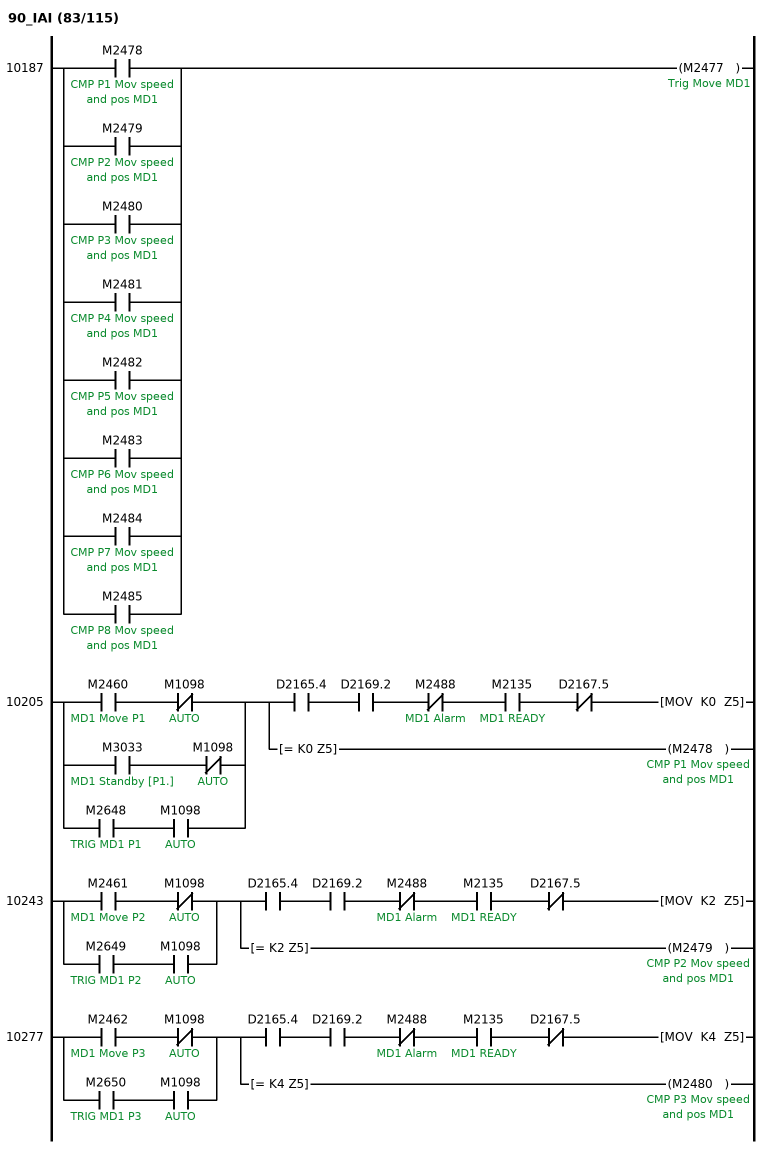
10187 LD      M2478  ; CMP P1 Mov speed and pos MD1
      OR      M2479  ; CMP P2 Mov speed and pos MD1
      OR      M2480  ; CMP P3 Mov speed and pos MD1
      OR      M2481  ; CMP P4 Mov speed and pos MD1
      OR      M2482  ; CMP P5 Mov speed and pos MD1
      OR      M2483  ; CMP P6 Mov speed and pos MD1
      OR      M2484  ; CMP P7 Mov speed and pos MD1
      OR      M2485  ; CMP P8 Mov speed and pos MD1
      OUT     M2477  ; Trig Move MD1
10205 LD      M2460  ; MD1 Move P1
      ANI     M1098  ; AUTO
      LD      M3033  ; MD1 Standby [P1.]
      ANI     M1098  ; AUTO
      ORB
      LD      M2648  ; TRIG MD1 P1
      AND     M1098  ; AUTO
      ORB
      MPS
      AND     D2165.4
      AND     D2169.2
      ANI     M2488  ; MD1 Alarm
      AND     M2135  ; MD1 READY
      ANI     D2167.5
      MOV     K0 Z5
      MPP
      AND=    K0 Z5
      OUT     M2478  ; CMP P1 Mov speed and pos MD1
10243 LD      M2461  ; MD1 Move P2
      ANI     M1098  ; AUTO
      LD      M2649  ; TRIG MD1 P2
      AND     M1098  ; AUTO
      ORB
      MPS
      AND     D2165.4
      AND     D2169.2
      ANI     M2488  ; MD1 Alarm
      AND     M2135  ; MD1 READY
      ANI     D2167.5
      MOV     K2 Z5
      MPP
      AND=    K2 Z5
      OUT     M2479  ; CMP P2 Mov speed and pos MD1
10277 LD      M2462  ; MD1 Move P3
      ANI     M1098  ; AUTO
      LD      M2650  ; TRIG MD1 P3
      AND     M1098  ; AUTO
      ORB
      MPS
      AND     D2165.4
      AND     D2169.2
      ANI     M2488  ; MD1 Alarm
      AND     M2135  ; MD1 READY
      ANI     D2167.5
      MOV     K4 Z5
      MPP
      AND=    K4 Z5
      OUT     M2480  ; CMP P3 Mov speed and pos MD1
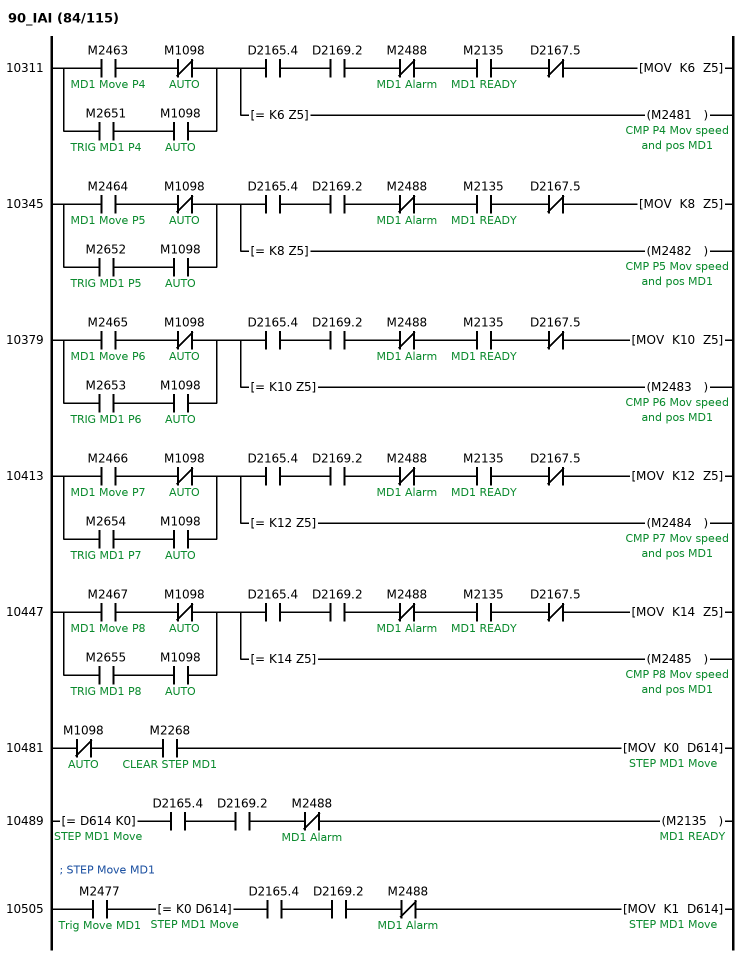
10311 LD      M2463  ; MD1 Move P4
      ANI     M1098  ; AUTO
      LD      M2651  ; TRIG MD1 P4
      AND     M1098  ; AUTO
      ORB
      MPS
      AND     D2165.4
      AND     D2169.2
      ANI     M2488  ; MD1 Alarm
      AND     M2135  ; MD1 READY
      ANI     D2167.5
      MOV     K6 Z5
      MPP
      AND=    K6 Z5
      OUT     M2481  ; CMP P4 Mov speed and pos MD1
10345 LD      M2464  ; MD1 Move P5
      ANI     M1098  ; AUTO
      LD      M2652  ; TRIG MD1 P5
      AND     M1098  ; AUTO
      ORB
      MPS
      AND     D2165.4
      AND     D2169.2
      ANI     M2488  ; MD1 Alarm
      AND     M2135  ; MD1 READY
      ANI     D2167.5
      MOV     K8 Z5
      MPP
      AND=    K8 Z5
      OUT     M2482  ; CMP P5 Mov speed and pos MD1
10379 LD      M2465  ; MD1 Move P6
      ANI     M1098  ; AUTO
      LD      M2653  ; TRIG MD1 P6
      AND     M1098  ; AUTO
      ORB
      MPS
      AND     D2165.4
      AND     D2169.2
      ANI     M2488  ; MD1 Alarm
      AND     M2135  ; MD1 READY
      ANI     D2167.5
      MOV     K10 Z5
      MPP
      AND=    K10 Z5
      OUT     M2483  ; CMP P6 Mov speed and pos MD1
10413 LD      M2466  ; MD1 Move P7
      ANI     M1098  ; AUTO
      LD      M2654  ; TRIG MD1 P7
      AND     M1098  ; AUTO
      ORB
      MPS
      AND     D2165.4
      AND     D2169.2
      ANI     M2488  ; MD1 Alarm
      AND     M2135  ; MD1 READY
      ANI     D2167.5
      MOV     K12 Z5
      MPP
      AND=    K12 Z5
      OUT     M2484  ; CMP P7 Mov speed and pos MD1
10447 LD      M2467  ; MD1 Move P8
      ANI     M1098  ; AUTO
      LD      M2655  ; TRIG MD1 P8
      AND     M1098  ; AUTO
      ORB
      MPS
      AND     D2165.4
      AND     D2169.2
      ANI     M2488  ; MD1 Alarm
      AND     M2135  ; MD1 READY
      ANI     D2167.5
      MOV     K14 Z5
      MPP
      AND=    K14 Z5
      OUT     M2485  ; CMP P8 Mov speed and pos MD1
10481 LDI     M1098  ; AUTO
      AND     M2268  ; CLEAR STEP MD1
      MOV     K0 D614
10489 LD=     D614 K0  ; STEP MD1 Move
      AND     D2165.4
      AND     D2169.2
      ANI     M2488  ; MD1 Alarm
      OUT     M2135  ; MD1 READY
; STEP Move MD1
10505 LD      M2477  ; Trig Move MD1
      AND=    K0 D614  ; STEP MD1 Move
      AND     D2165.4
      AND     D2169.2
      ANI     M2488  ; MD1 Alarm
      MOV     K1 D614
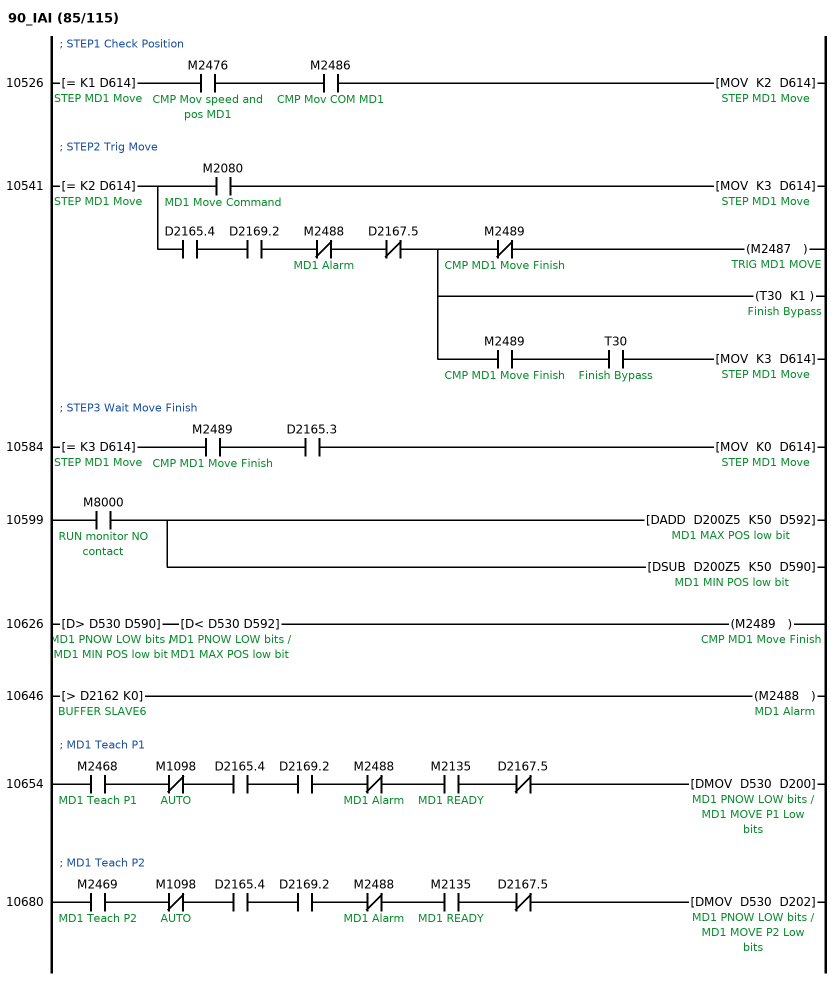
; STEP1 Check Position
10526 LD=     K1 D614  ; STEP MD1 Move
      AND     M2476  ; CMP Mov speed and pos MD1
      AND     M2486  ; CMP Mov COM MD1
      MOV     K2 D614
; STEP2 Trig Move
10541 LD=     K2 D614  ; STEP MD1 Move
      MPS
      AND     M2080  ; MD1 Move Command
      MOV     K3 D614
      MPP
      AND     D2165.4
      AND     D2169.2
      ANI     M2488  ; MD1 Alarm
      ANI     D2167.5
      MPS
      ANI     M2489  ; CMP MD1 Move Finish
      OUT     M2487  ; TRIG MD1 MOVE
      MPP
      OUT     T30 K1  ; Finish Bypass
      AND     M2489  ; CMP MD1 Move Finish
      AND     T30  ; Finish Bypass
      MOV     K3 D614
; STEP3 Wait Move Finish
10584 LD=     K3 D614  ; STEP MD1 Move
      AND     M2489  ; CMP MD1 Move Finish
      AND     D2165.3
      MOV     K0 D614
10599 LD      M8000  ; RUN monitor NO contact
      DADD    D200Z5 K50 D592  ; MD1 MAX POS low bit
      DSUB    D200Z5 K50 D590  ; MD1 MIN POS low bit
10626 LDD>    D530 D590  ; MD1 PNOW LOW bits / MD1 MIN POS low bit
      ANDD<   D530 D592  ; MD1 PNOW LOW bits / MD1 MAX POS low bit
      OUT     M2489  ; CMP MD1 Move Finish
10646 LD>     D2162 K0  ; BUFFER SLAVE6
      OUT     M2488  ; MD1 Alarm
; MD1 Teach P1
10654 LD      M2468  ; MD1 Teach P1
      ANI     M1098  ; AUTO
      AND     D2165.4
      AND     D2169.2
      ANI     M2488  ; MD1 Alarm
      AND     M2135  ; MD1 READY
      ANI     D2167.5
      DMOV    D530 D200  ; MD1 MOVE P1 Low bits
; MD1 Teach P2
10680 LD      M2469  ; MD1 Teach P2
      ANI     M1098  ; AUTO
      AND     D2165.4
      AND     D2169.2
      ANI     M2488  ; MD1 Alarm
      AND     M2135  ; MD1 READY
      ANI     D2167.5
      DMOV    D530 D202  ; MD1 MOVE P2 Low bits
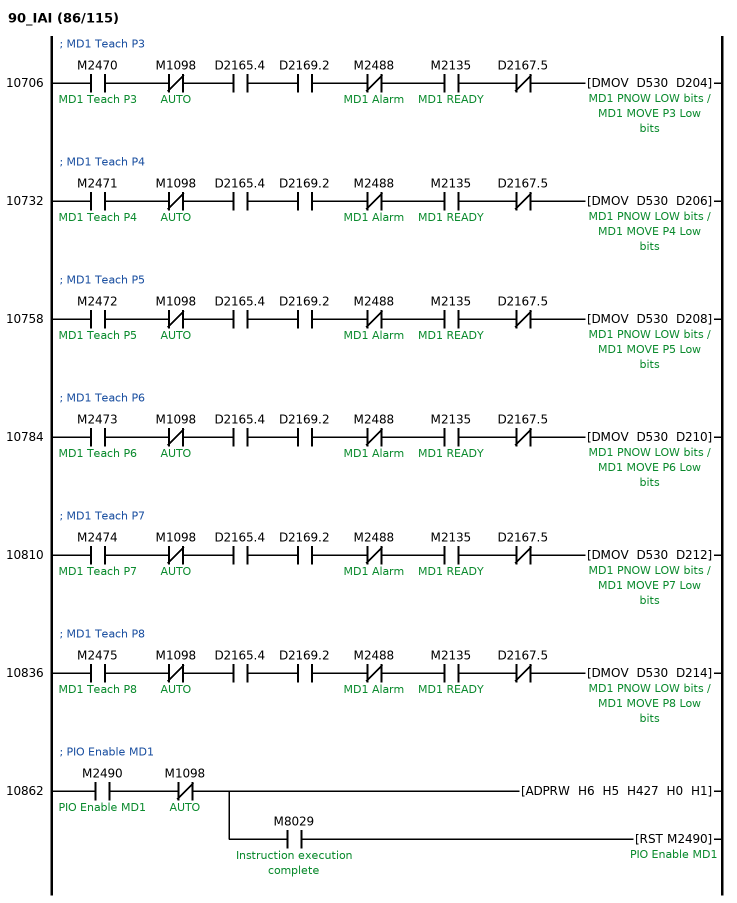
; MD1 Teach P3
10706 LD      M2470  ; MD1 Teach P3
      ANI     M1098  ; AUTO
      AND     D2165.4
      AND     D2169.2
      ANI     M2488  ; MD1 Alarm
      AND     M2135  ; MD1 READY
      ANI     D2167.5
      DMOV    D530 D204  ; MD1 MOVE P3 Low bits
; MD1 Teach P4
10732 LD      M2471  ; MD1 Teach P4
      ANI     M1098  ; AUTO
      AND     D2165.4
      AND     D2169.2
      ANI     M2488  ; MD1 Alarm
      AND     M2135  ; MD1 READY
      ANI     D2167.5
      DMOV    D530 D206  ; MD1 MOVE P4 Low bits
; MD1 Teach P5
10758 LD      M2472  ; MD1 Teach P5
      ANI     M1098  ; AUTO
      AND     D2165.4
      AND     D2169.2
      ANI     M2488  ; MD1 Alarm
      AND     M2135  ; MD1 READY
      ANI     D2167.5
      DMOV    D530 D208  ; MD1 MOVE P5 Low bits
; MD1 Teach P6
10784 LD      M2473  ; MD1 Teach P6
      ANI     M1098  ; AUTO
      AND     D2165.4
      AND     D2169.2
      ANI     M2488  ; MD1 Alarm
      AND     M2135  ; MD1 READY
      ANI     D2167.5
      DMOV    D530 D210  ; MD1 MOVE P6 Low bits
; MD1 Teach P7
10810 LD      M2474  ; MD1 Teach P7
      ANI     M1098  ; AUTO
      AND     D2165.4
      AND     D2169.2
      ANI     M2488  ; MD1 Alarm
      AND     M2135  ; MD1 READY
      ANI     D2167.5
      DMOV    D530 D212  ; MD1 MOVE P7 Low bits
; MD1 Teach P8
10836 LD      M2475  ; MD1 Teach P8
      ANI     M1098  ; AUTO
      AND     D2165.4
      AND     D2169.2
      ANI     M2488  ; MD1 Alarm
      AND     M2135  ; MD1 READY
      ANI     D2167.5
      DMOV    D530 D214  ; MD1 MOVE P8 Low bits
; PIO Enable MD1
10862 LD      M2490  ; PIO Enable MD1
      ANI     M1098  ; AUTO
      ADPRW   H6 H5 H427 H0 H1
      AND     M8029  ; Instruction execution complete
      RST     M2490  ; PIO Enable MD1
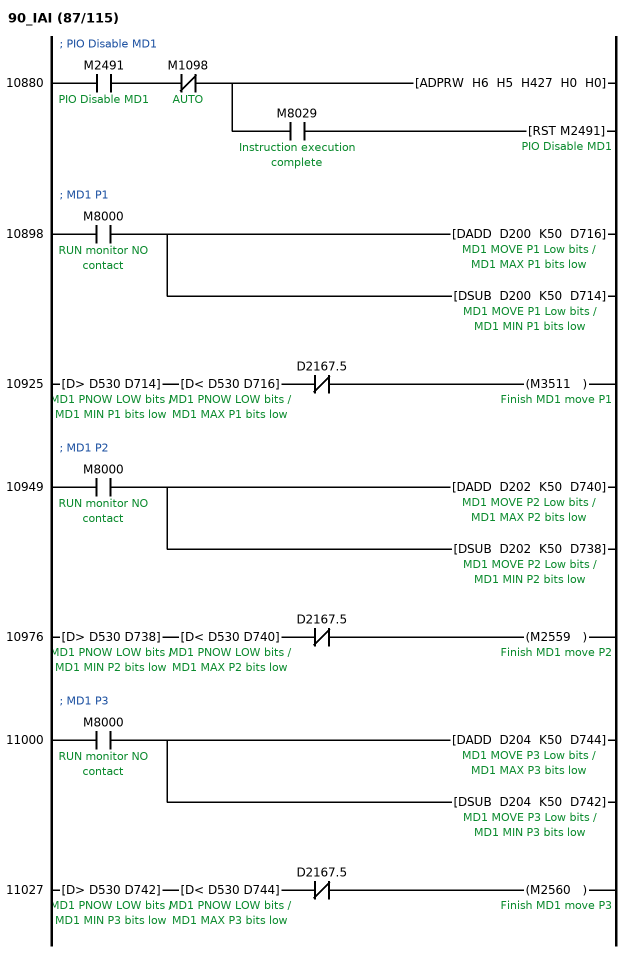
; PIO Disable MD1
10880 LD      M2491  ; PIO Disable MD1
      ANI     M1098  ; AUTO
      ADPRW   H6 H5 H427 H0 H0
      AND     M8029  ; Instruction execution complete
      RST     M2491  ; PIO Disable MD1
; MD1 P1
10898 LD      M8000  ; RUN monitor NO contact
      DADD    D200 K50 D716  ; MD1 MAX P1 bits low
      DSUB    D200 K50 D714  ; MD1 MIN P1 bits low
10925 LDD>    D530 D714  ; MD1 PNOW LOW bits / MD1 MIN P1 bits low
      ANDD<   D530 D716  ; MD1 PNOW LOW bits / MD1 MAX P1 bits low
      ANI     D2167.5
      OUT     M3511  ; Finish MD1 move P1
; MD1 P2
10949 LD      M8000  ; RUN monitor NO contact
      DADD    D202 K50 D740  ; MD1 MAX P2 bits low
      DSUB    D202 K50 D738  ; MD1 MIN P2 bits low
10976 LDD>    D530 D738  ; MD1 PNOW LOW bits / MD1 MIN P2 bits low
      ANDD<   D530 D740  ; MD1 PNOW LOW bits / MD1 MAX P2 bits low
      ANI     D2167.5
      OUT     M2559  ; Finish MD1 move P2
; MD1 P3
11000 LD      M8000  ; RUN monitor NO contact
      DADD    D204 K50 D744  ; MD1 MAX P3 bits low
      DSUB    D204 K50 D742  ; MD1 MIN P3 bits low
11027 LDD>    D530 D742  ; MD1 PNOW LOW bits / MD1 MIN P3 bits low
      ANDD<   D530 D744  ; MD1 PNOW LOW bits / MD1 MAX P3 bits low
      ANI     D2167.5
      OUT     M2560  ; Finish MD1 move P3
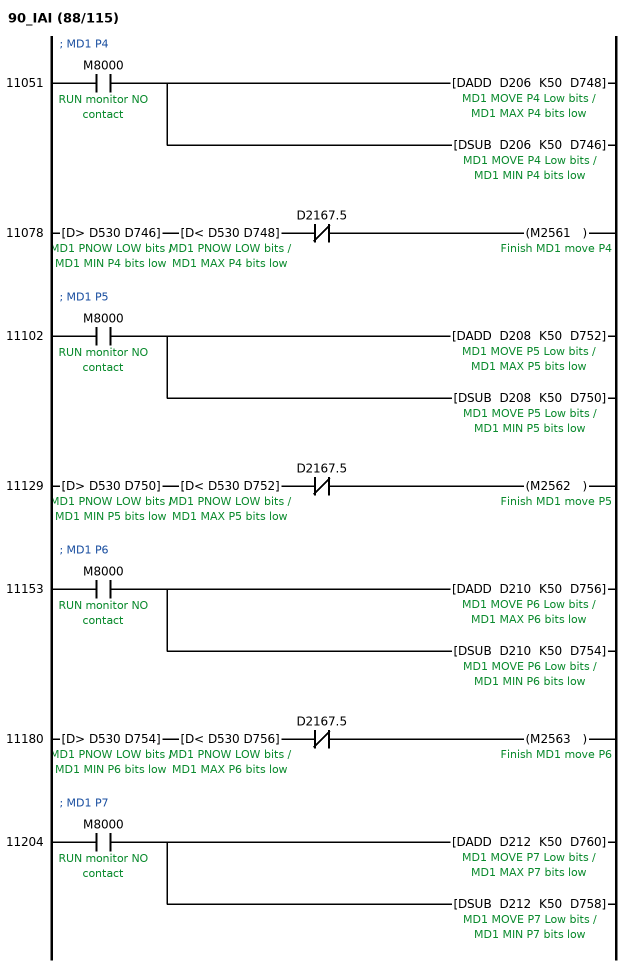
; MD1 P4
11051 LD      M8000  ; RUN monitor NO contact
      DADD    D206 K50 D748  ; MD1 MAX P4 bits low
      DSUB    D206 K50 D746  ; MD1 MIN P4 bits low
11078 LDD>    D530 D746  ; MD1 PNOW LOW bits / MD1 MIN P4 bits low
      ANDD<   D530 D748  ; MD1 PNOW LOW bits / MD1 MAX P4 bits low
      ANI     D2167.5
      OUT     M2561  ; Finish MD1 move P4
; MD1 P5
11102 LD      M8000  ; RUN monitor NO contact
      DADD    D208 K50 D752  ; MD1 MAX P5 bits low
      DSUB    D208 K50 D750  ; MD1 MIN P5 bits low
11129 LDD>    D530 D750  ; MD1 PNOW LOW bits / MD1 MIN P5 bits low
      ANDD<   D530 D752  ; MD1 PNOW LOW bits / MD1 MAX P5 bits low
      ANI     D2167.5
      OUT     M2562  ; Finish MD1 move P5
; MD1 P6
11153 LD      M8000  ; RUN monitor NO contact
      DADD    D210 K50 D756  ; MD1 MAX P6 bits low
      DSUB    D210 K50 D754  ; MD1 MIN P6 bits low
11180 LDD>    D530 D754  ; MD1 PNOW LOW bits / MD1 MIN P6 bits low
      ANDD<   D530 D756  ; MD1 PNOW LOW bits / MD1 MAX P6 bits low
      ANI     D2167.5
      OUT     M2563  ; Finish MD1 move P6
; MD1 P7
11204 LD      M8000  ; RUN monitor NO contact
      DADD    D212 K50 D760  ; MD1 MAX P7 bits low
      DSUB    D212 K50 D758  ; MD1 MIN P7 bits low
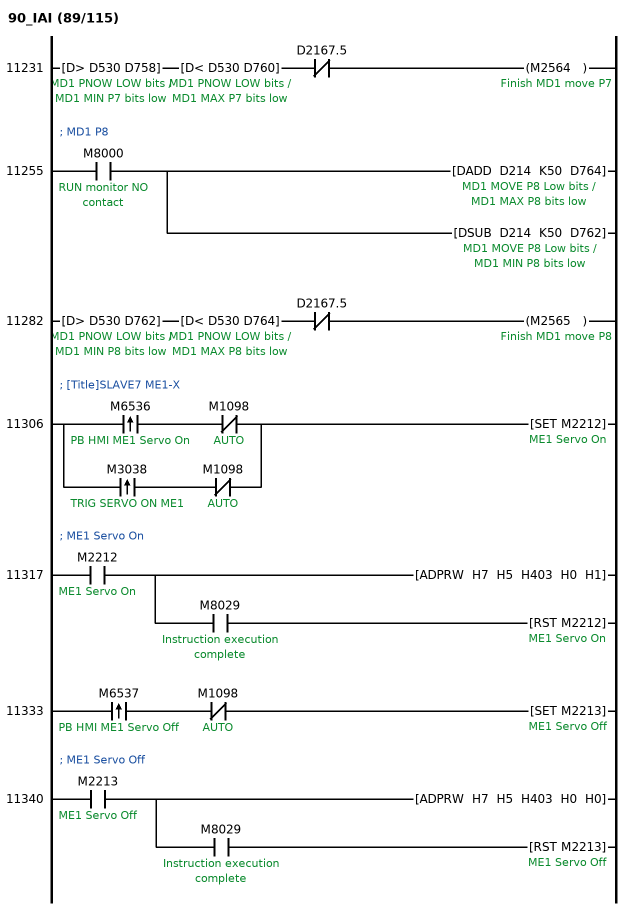
11231 LDD>    D530 D758  ; MD1 PNOW LOW bits / MD1 MIN P7 bits low
      ANDD<   D530 D760  ; MD1 PNOW LOW bits / MD1 MAX P7 bits low
      ANI     D2167.5
      OUT     M2564  ; Finish MD1 move P7
; MD1 P8
11255 LD      M8000  ; RUN monitor NO contact
      DADD    D214 K50 D764  ; MD1 MAX P8 bits low
      DSUB    D214 K50 D762  ; MD1 MIN P8 bits low
11282 LDD>    D530 D762  ; MD1 PNOW LOW bits / MD1 MIN P8 bits low
      ANDD<   D530 D764  ; MD1 PNOW LOW bits / MD1 MAX P8 bits low
      ANI     D2167.5
      OUT     M2565  ; Finish MD1 move P8
; [Title]SLAVE7 ME1-X
11306 LDP     M6536  ; PB HMI ME1 Servo On
      ANI     M1098  ; AUTO
      LDP     M3038  ; TRIG SERVO ON ME1
      ANI     M1098  ; AUTO
      ORB
      SET     M2212  ; ME1 Servo On
; ME1 Servo On
11317 LD      M2212  ; ME1 Servo On
      ADPRW   H7 H5 H403 H0 H1
      AND     M8029  ; Instruction execution complete
      RST     M2212  ; ME1 Servo On
11333 LDP     M6537  ; PB HMI ME1 Servo Off
      ANI     M1098  ; AUTO
      SET     M2213  ; ME1 Servo Off
; ME1 Servo Off
11340 LD      M2213  ; ME1 Servo Off
      ADPRW   H7 H5 H403 H0 H0
      AND     M8029  ; Instruction execution complete
      RST     M2213  ; ME1 Servo Off
